// TIA Portal V19 export
DATA_BLOCK "Main_Safety_RTG1_DB"   // DB18, F_DB
// stored: AutoNumber false, InstanceOfName Main_Safety_RTG1, InstanceOfType FB
"Main_Safety_RTG1"
BEGIN
END_DATA_BLOCK
